FUNCTION_BLOCK IO_DQ32 (* Cartao TM3DQ32TK da remota TM3BCEIP: le 32 comandos BOOL por symlink e escreve as 2 words na remota sempre (sem bloqueio por comunicacao), com depurador *)
  (* Standard: 61499-2 *)
  (* Version 1.1, 10/6/2026, Hidryco, Hidryco, 1.1: removido o gate de comunicacao; escrita nunca depende do status da remota *)
  PACKAGE Hidryco.HidrycoLib;
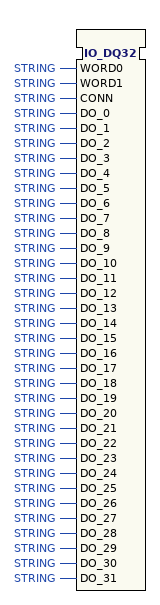
  VAR_INPUT
    WORD0 : STRING; (* Nome do symlink da word 0 do cartao (bits 0-15), ex.: A7_Q0_0_15 *)
    WORD1 : STRING; (* Nome do symlink da word 1 do cartao (bits 16-31) *)
    CONN : STRING; (* Opcional, so diagnostico no depurador: symlink connStatusInt da remota. NAO interfere na escrita das saidas *)
    DO_0 : STRING; (* Nome do symlink BOOL lido como comando do bit 0 do cartao *)
    DO_1 : STRING; (* Nome do symlink BOOL lido como comando do bit 1 do cartao *)
    DO_2 : STRING; (* Nome do symlink BOOL lido como comando do bit 2 do cartao *)
    DO_3 : STRING; (* Nome do symlink BOOL lido como comando do bit 3 do cartao *)
    DO_4 : STRING; (* Nome do symlink BOOL lido como comando do bit 4 do cartao *)
    DO_5 : STRING; (* Nome do symlink BOOL lido como comando do bit 5 do cartao *)
    DO_6 : STRING; (* Nome do symlink BOOL lido como comando do bit 6 do cartao *)
    DO_7 : STRING; (* Nome do symlink BOOL lido como comando do bit 7 do cartao *)
    DO_8 : STRING; (* Nome do symlink BOOL lido como comando do bit 8 do cartao *)
    DO_9 : STRING; (* Nome do symlink BOOL lido como comando do bit 9 do cartao *)
    DO_10 : STRING; (* Nome do symlink BOOL lido como comando do bit 10 do cartao *)
    DO_11 : STRING; (* Nome do symlink BOOL lido como comando do bit 11 do cartao *)
    DO_12 : STRING; (* Nome do symlink BOOL lido como comando do bit 12 do cartao *)
    DO_13 : STRING; (* Nome do symlink BOOL lido como comando do bit 13 do cartao *)
    DO_14 : STRING; (* Nome do symlink BOOL lido como comando do bit 14 do cartao *)
    DO_15 : STRING; (* Nome do symlink BOOL lido como comando do bit 15 do cartao *)
    DO_16 : STRING; (* Nome do symlink BOOL lido como comando do bit 16 do cartao *)
    DO_17 : STRING; (* Nome do symlink BOOL lido como comando do bit 17 do cartao *)
    DO_18 : STRING; (* Nome do symlink BOOL lido como comando do bit 18 do cartao *)
    DO_19 : STRING; (* Nome do symlink BOOL lido como comando do bit 19 do cartao *)
    DO_20 : STRING; (* Nome do symlink BOOL lido como comando do bit 20 do cartao *)
    DO_21 : STRING; (* Nome do symlink BOOL lido como comando do bit 21 do cartao *)
    DO_22 : STRING; (* Nome do symlink BOOL lido como comando do bit 22 do cartao *)
    DO_23 : STRING; (* Nome do symlink BOOL lido como comando do bit 23 do cartao *)
    DO_24 : STRING; (* Nome do symlink BOOL lido como comando do bit 24 do cartao *)
    DO_25 : STRING; (* Nome do symlink BOOL lido como comando do bit 25 do cartao *)
    DO_26 : STRING; (* Nome do symlink BOOL lido como comando do bit 26 do cartao *)
    DO_27 : STRING; (* Nome do symlink BOOL lido como comando do bit 27 do cartao *)
    DO_28 : STRING; (* Nome do symlink BOOL lido como comando do bit 28 do cartao *)
    DO_29 : STRING; (* Nome do symlink BOOL lido como comando do bit 29 do cartao *)
    DO_30 : STRING; (* Nome do symlink BOOL lido como comando do bit 30 do cartao *)
    DO_31 : STRING; (* Nome do symlink BOOL lido como comando do bit 31 do cartao *)
  END_VAR
  FBS
    plcStart1 : plcStart(Prio := 3);
    IThis : IO_DQ32_HMI(QI := TRUE);
    DST_CONN : SYMLINKMULTIVARDST_5A03F112CD5D470(QI := TRUE); {SET_ATTRIBUTE(Configuration.GenericFBType.InterfaceParams, Runtime.System#I:=1;VALUE${I$}:INT)}
    DST_B0 : SYMLINKMULTIVARDST_854A896E88500D19(QI := TRUE); {SET_ATTRIBUTE(Configuration.GenericFBType.InterfaceParams, Runtime.System#I:=16;VALUE${I$}:BOOL,BOOL,BOOL,BOOL,BOOL,BOOL,BOOL,BOOL,BOOL,BOOL,BOOL,BOOL,BOOL,BOOL,BOOL,BOOL)}
    PACK_0 : BITMAN_182F748F2FAD4D59; {SET_ATTRIBUTE(Configuration.GenericFBType.InterfaceParams, Runtime.Standard#CNTIN:=16;CNTOUT:=1;IN${CNTIN$}:BOOL,BOOL,BOOL,BOOL,BOOL,BOOL,BOOL,BOOL,BOOL,BOOL,BOOL,BOOL,BOOL,BOOL,BOOL,BOOL;OUT${CNTOUT$}:WORD)}
    W2I_0 : ANY2ANY_200292F8C654761DB; {SET_ATTRIBUTE(Configuration.GenericFBType.InterfaceParams, Runtime.Standard#CNT:=1;IN${CNT$}:WORD;OUT${CNT$}:INT)}
    SRC_W0 : SYMLINKMULTIVARSRC_5A03F112CD5D470(QI := TRUE); {SET_ATTRIBUTE(Configuration.GenericFBType.InterfaceParams, Runtime.System#I:=1;VALUE${I$}:INT)}
    DST_B1 : SYMLINKMULTIVARDST_854A896E88500D19(QI := TRUE); {SET_ATTRIBUTE(Configuration.GenericFBType.InterfaceParams, Runtime.System#I:=16;VALUE${I$}:BOOL,BOOL,BOOL,BOOL,BOOL,BOOL,BOOL,BOOL,BOOL,BOOL,BOOL,BOOL,BOOL,BOOL,BOOL,BOOL)}
    PACK_1 : BITMAN_182F748F2FAD4D59; {SET_ATTRIBUTE(Configuration.GenericFBType.InterfaceParams, Runtime.Standard#CNTIN:=16;CNTOUT:=1;IN${CNTIN$}:BOOL,BOOL,BOOL,BOOL,BOOL,BOOL,BOOL,BOOL,BOOL,BOOL,BOOL,BOOL,BOOL,BOOL,BOOL,BOOL;OUT${CNTOUT$}:WORD)}
    W2I_1 : ANY2ANY_200292F8C654761DB; {SET_ATTRIBUTE(Configuration.GenericFBType.InterfaceParams, Runtime.Standard#CNT:=1;IN${CNT$}:WORD;OUT${CNT$}:INT)}
    SRC_W1 : SYMLINKMULTIVARSRC_5A03F112CD5D470(QI := TRUE); {SET_ATTRIBUTE(Configuration.GenericFBType.InterfaceParams, Runtime.System#I:=1;VALUE${I$}:INT)}
  END_FBS
  EVENT_CONNECTIONS
    DST_B0.CNF TO PACK_0.REQ;
    PACK_0.CNF TO W2I_0.REQ;
    W2I_0.CNF TO SRC_W0.REQ;
    DST_B1.CNF TO PACK_1.REQ;
    PACK_1.CNF TO W2I_1.REQ;
    W2I_1.CNF TO SRC_W1.REQ;
    plcStart1.FIRST_INIT TO DST_B0.INIT;
    plcStart1.REDO_INIT TO DST_B0.INIT;
    DST_B0.INITO TO DST_B1.INIT;
    DST_B1.INITO TO DST_CONN.INIT;
    DST_CONN.INITO TO PACK_0.INIT;
    PACK_0.INITO TO PACK_1.INIT;
    PACK_1.INITO TO SRC_W0.INIT;
    SRC_W0.INITO TO SRC_W1.INIT;
    SRC_W1.INITO TO IThis.2580331DF766B7BD;
    IThis.B2F0B7003C60D222 TO plcStart1.ACK_FIRST;
    W2I_0.CNF TO IThis.C93D1AB5D9425049;
    W2I_1.CNF TO IThis.C93D1AB5D9425049;
    DST_CONN.CNF TO IThis.C93D1AB5D9425049;
  END_CONNECTIONS
  DATA_CONNECTIONS
    PACK_0.OUT1 TO W2I_0.IN1;
    W2I_0.OUT1 TO SRC_W0.VALUE1;
    WORD0 TO SRC_W0.NAME1;
    W2I_0.OUT1 TO IThis.3A722DFD35FBCED2;
    DST_B0.VALUE1 TO PACK_0.IN1;
    DST_B0.VALUE1 TO IThis.03F32C95190C8373;
    DO_0 TO DST_B0.NAME1;
    DST_B0.VALUE2 TO PACK_0.IN2;
    DST_B0.VALUE2 TO IThis.BCF96A408D99644D;
    DO_1 TO DST_B0.NAME2;
    DST_B0.VALUE3 TO PACK_0.IN3;
    DST_B0.VALUE3 TO IThis.FAD9B6BA1A6CC0D0;
    DO_2 TO DST_B0.NAME3;
    DST_B0.VALUE4 TO PACK_0.IN4;
    DST_B0.VALUE4 TO IThis.E3DA1A4F68587796;
    DO_3 TO DST_B0.NAME4;
    DST_B0.VALUE5 TO PACK_0.IN5;
    DST_B0.VALUE5 TO IThis.9A745A6FFBA842D7;
    DO_4 TO DST_B0.NAME5;
    DST_B0.VALUE6 TO PACK_0.IN6;
    DST_B0.VALUE6 TO IThis.A2C27D279617865B;
    DO_5 TO DST_B0.NAME6;
    DST_B0.VALUE7 TO PACK_0.IN7;
    DST_B0.VALUE7 TO IThis.DD025B0B81756BA3;
    DO_6 TO DST_B0.NAME7;
    DST_B0.VALUE8 TO PACK_0.IN8;
    DST_B0.VALUE8 TO IThis.4D8CA11CED3C30FF;
    DO_7 TO DST_B0.NAME8;
    DST_B0.VALUE9 TO PACK_0.IN9;
    DST_B0.VALUE9 TO IThis.4F8132BA8F6FA096;
    DO_8 TO DST_B0.NAME9;
    DST_B0.VALUE10 TO PACK_0.IN10;
    DST_B0.VALUE10 TO IThis.563F82C8E47B7F5C;
    DO_9 TO DST_B0.NAME10;
    DST_B0.VALUE11 TO PACK_0.IN11;
    DST_B0.VALUE11 TO IThis.FDA5BE9A9817ACCB;
    DO_10 TO DST_B0.NAME11;
    DST_B0.VALUE12 TO PACK_0.IN12;
    DST_B0.VALUE12 TO IThis.20FDDC1F0E800049;
    DO_11 TO DST_B0.NAME12;
    DST_B0.VALUE13 TO PACK_0.IN13;
    DST_B0.VALUE13 TO IThis.FFCD8534758C21C7;
    DO_12 TO DST_B0.NAME13;
    DST_B0.VALUE14 TO PACK_0.IN14;
    DST_B0.VALUE14 TO IThis.B093681444B02D5E;
    DO_13 TO DST_B0.NAME14;
    DST_B0.VALUE15 TO PACK_0.IN15;
    DST_B0.VALUE15 TO IThis.0372E9569935B60A;
    DO_14 TO DST_B0.NAME15;
    DST_B0.VALUE16 TO PACK_0.IN16;
    DST_B0.VALUE16 TO IThis.E99A35F7ED61F737;
    DO_15 TO DST_B0.NAME16;
    PACK_1.OUT1 TO W2I_1.IN1;
    W2I_1.OUT1 TO SRC_W1.VALUE1;
    WORD1 TO SRC_W1.NAME1;
    W2I_1.OUT1 TO IThis.3D7D13936729667D;
    DST_B1.VALUE1 TO PACK_1.IN1;
    DST_B1.VALUE1 TO IThis.3436F174B0C6DB0A;
    DO_16 TO DST_B1.NAME1;
    DST_B1.VALUE2 TO PACK_1.IN2;
    DST_B1.VALUE2 TO IThis.1DF5DA3794E56E35;
    DO_17 TO DST_B1.NAME2;
    DST_B1.VALUE3 TO PACK_1.IN3;
    DST_B1.VALUE3 TO IThis.1B89BF053C4711E9;
    DO_18 TO DST_B1.NAME3;
    DST_B1.VALUE4 TO PACK_1.IN4;
    DST_B1.VALUE4 TO IThis.25866A3ADFE41BAD;
    DO_19 TO DST_B1.NAME4;
    DST_B1.VALUE5 TO PACK_1.IN5;
    DST_B1.VALUE5 TO IThis.0D4A9E3E56E9E60A;
    DO_20 TO DST_B1.NAME5;
    DST_B1.VALUE6 TO PACK_1.IN6;
    DST_B1.VALUE6 TO IThis.518F4858C5D2F237;
    DO_21 TO DST_B1.NAME6;
    DST_B1.VALUE7 TO PACK_1.IN7;
    DST_B1.VALUE7 TO IThis.A6C6760779C9B21A;
    DO_22 TO DST_B1.NAME7;
    DST_B1.VALUE8 TO PACK_1.IN8;
    DST_B1.VALUE8 TO IThis.CB0E5882CB7E2035;
    DO_23 TO DST_B1.NAME8;
    DST_B1.VALUE9 TO PACK_1.IN9;
    DST_B1.VALUE9 TO IThis.FD3F0F4D41A840BA;
    DO_24 TO DST_B1.NAME9;
    DST_B1.VALUE10 TO PACK_1.IN10;
    DST_B1.VALUE10 TO IThis.8B41E1BD56994A18;
    DO_25 TO DST_B1.NAME10;
    DST_B1.VALUE11 TO PACK_1.IN11;
    DST_B1.VALUE11 TO IThis.C76414CB004EACB4;
    DO_26 TO DST_B1.NAME11;
    DST_B1.VALUE12 TO PACK_1.IN12;
    DST_B1.VALUE12 TO IThis.FBA6993DCAE315B7;
    DO_27 TO DST_B1.NAME12;
    DST_B1.VALUE13 TO PACK_1.IN13;
    DST_B1.VALUE13 TO IThis.4BC433EFA713E10C;
    DO_28 TO DST_B1.NAME13;
    DST_B1.VALUE14 TO PACK_1.IN14;
    DST_B1.VALUE14 TO IThis.216747715E093DEF;
    DO_29 TO DST_B1.NAME14;
    DST_B1.VALUE15 TO PACK_1.IN15;
    DST_B1.VALUE15 TO IThis.A1A3BEA4372BFC0F;
    DO_30 TO DST_B1.NAME15;
    DST_B1.VALUE16 TO PACK_1.IN16;
    DST_B1.VALUE16 TO IThis.FCE742B05E32D725;
    DO_31 TO DST_B1.NAME16;
    CONN TO DST_CONN.NAME1;
    DST_CONN.VALUE1 TO IThis.750DA6EE7F1E02B1;
  END_CONNECTIONS
END_FUNCTION_BLOCK
